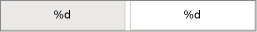
VISUALIZATION VISU_ConfigUSINTEntry  // 257x32
VAR_IN_OUT
    active : USINT;
    editable : USINT;
END_VAR
    Textfield (0,0 125x30), "%d", text variable: active, input disabled if: TRUE
    Textfield (130,0 125x30), "%d", text variable: editable, colour toggle: editable <> active
        OnMouseClick: write the text variable via Default
END_VISUALIZATION

(* stored: Version 1.1.0.1, ProductVersion 3.1.0.36
   Visu VISU_ConfigUSINTEntry: Id {111eddce-8ada-4c21-bba3-952eb91722d9} *)
